FUNCTION F_BYTE_TO_REAL : REAL
VAR_INPUT
    BY1 : BYTE;
    BY2 : BYTE;
    BY3 : BYTE;
    BY4 : BYTE;
END_VAR
VAR
   OutVAR : DWORD; 
   OutVarREAL : REAL;
END_VAR

OutVar := BY1;
OutVar := SHL(OutVar, 8) OR BY2;
OutVar := SHL(OutVar, 8) OR BY3;
OutVar := SHL(OutVar, 8) OR BY4;

MEMCPY(ADR(OutVarREAL), ADR(OutVar), SIZEOF(REAL));
F_BYTE_TO_REAL := OutVarREAL;

END_FUNCTION

(* stored: Version 1.1.0.1
   POU F_BYTE_TO_REAL: Id {03556380-be63-4ca9-82d4-6199857e8d87}, SpecialFunc None *)
